FUNCTION_BLOCK StrapMachineOld
VAR
	manual : BOOL; //:= TRUE;
	
	error AT %I* : BOOL;
	ready AT %I* : BOOL;
	//busy AT %I* : BOOL;
	done AT %I* : BOOL;
	home AT %I* : BOOL;
	
	execute AT %Q* : BOOL;
	enable AT %Q* : BOOL;
	reset AT %Q* : BOOL;

	start : BOOL;
	
	timeout : TON;
	hold : TON;
	
	step : (SETUP, STRAP, WAIT);
	
	i : INT;
END_VAR
VAR CONSTANT
	pulseWidth : TIME := T#500MS;
	delayTime : TIME := T#500MS;
	
	failTime : TIME := T#30S;
END_VAR

hold(IN:= , PT:= delayTime, Q=> , ET=> );
timeout(IN:= step > SETUP, PT:= failTime, Q=> , ET=> );

IF timeout.Q THEN
	timeout.IN := FALSE;
	step := SETUP;
END_IF

IF manual THEN
	RETURN;
END_IF

CASE step OF	
	SETUP:
		IF NOT error THEN
			reset := FALSE;
			enable := TRUE;
			
			IF start THEN
				start := FALSE;
				step := STRAP;
			END_IF
			
		ELSE
			reset := NOT reset;
			enable := NOT enable;
		END_IF
	
	STRAP:
		IF NOT execute THEN
			execute := TRUE;
			RETURN;
		END_IF
		
		IF execute AND NOT home THEN
			execute := FALSE;
			step := WAIT;
		END_IF
		
	WAIT:
		IF home THEN
			hold.IN := TRUE;
			enable := FALSE;
			execute := FALSE;
		END_IF
		
		IF hold.Q THEN
			hold.IN := FALSE;
			i := i + 1;
			step := 0;			
		END_IF
END_CASE

END_FUNCTION_BLOCK

(* stored: Version 1.1.0.1, ProductVersion 3.1.4024.12
   POU StrapMachineOld: Id {b80a0c4b-c6af-42e3-9ea6-1e5c8f9c9f0a}, SpecialFunc None *)
